Fanuc KAREL source: ks00048.KL

PROGRAM KS00048
%STACKSIZE=65535
%PRIORITY=65535
%NOLOCKGROUP
VAR
A : ARRAY[4] OF XYZWPREXT
B : ARRAY[4] OF XYZWPREXT
FLAG : BOOLEAN
N : INTEGER
STATUS : INTEGER
PN : STRING[80]
VN : STRING[80]
BEGIN
PN=''
VN='A'
-- UNRESOLVED_PC line 19 opcodes [27 22 22 2A 22 2A 22 22 AF] marker_code=27
END KS00048
